FUNCTION_BLOCK FB_Logger IMPLEMENTS ZigasLibs_Core.I_LoggerEx
VAR
	_fileProperties			: ST_FileProperties;
	_logLevelHeaders		: ZigasLibs_Core.ST_LogLevelHeaders;
	_fileHandler			: FB_FileHandler;
	_logEntries				: ARRAY[0..100] OF Tc2_System.T_MaxString;
	_state					: E_LoggerState;
	_oldState				: E_LoggerState;
	_fileExists				: BOOL;
	_localSystemTime		: ZigasLibs_Core.FB_LocalSystemTimeProvider;
	_localSystemTimeString	: Tc2_System.T_MaxString;
	_stringBuilder			: ZigasLibs_Core.FB_StringBuilderBase;
	_amsAddress				: Tc2_System.ST_AmsAddr;
	_dateForLogName			: STRING;
END_VAR

_localSystemTime();
_localSystemTimeString := _localSystemTime.ConvertToString()
	.DateTime(dateSeperator := '.',
		fillWithZeros := TRUE,
		IncludeMilliseconds := FALSE,
		timeFormat := ZigasLibs_Core.E_TimeFormat.YYMMDD_HHMMSS,
		timeOfDaySeperator := ':');

IF _fileHandler.Error THEN
	_state := E_LoggerState.Error;
END_IF

CASE _state OF 
	E_LoggerState.IDLE:
		IF _logEntries[0] <> '' AND _localSystemTime.CurrentTime.IsValid THEN
			_state := E_LoggerState.WRITE_TO_FILE;
		END_IF		
		
	E_LoggerState.WRITE_TO_FILE:
		_fileHandler.FileProperties.FileLocation := _fileProperties.FileLocation;
		_fileHandler.AmsAddress.netId := AmsAddress.netId;
		_dateForLogName := _localSystemTime.ConvertToString().DateTime(
			timeFormat := ZigasLibs_Core.E_TimeFormat.YYMMDD,
			timeOfDaySeperator := '',
			dateSeperator := '',
			fillWithZeros := TRUE,
			IncludeMilliseconds := FALSE);

		_dateForLogName := _stringBuilder.Reset()
			.AddString(str := _dateForLogName)
			.AddString(str := '_')
			.AddString(str := _localSystemTime.ConvertToString().Hour(fillWithZeros := TRUE))
			.Create();
	
		_fileHandler.FileProperties.FileName := _stringBuilder.Reset()
			.AddString(str := _fileProperties.FileName)
			.AddString(str := '_')
			.AddString(str := _dateForLogName)
			.AddString(str := '.txt')
			.Create();
		
		IF NOT _fileHandler.Error AND_THEN 
			_fileHandler.WriteLine_Append(sContent := _logEntries[0]) 
		THEN
			RemoveLogEntry();
			_state := E_LoggerState.IDLE;
		END_IF
		
	E_LoggerState.ERROR:
		IF _oldState <> E_LoggerState.ERROR THEN
			_fileHandler.Reset();
		END_IF
END_CASE

_oldState := _state;

METHOD PRIVATE AddLogEntry
VAR_INPUT
	message	: Tc2_System.T_MaxString;
END_VAR

VAR
	i				: ZigasLibs_Core.T_ArrayIndexer;
	eventsMaxIndex	: ZigasLibs_Core.T_ArrayIndexer;
END_VAR
message := Tc2_Standard.CONCAT(
	STR1 := message, 
	STR2 := ZigasLibs_Core.StringConstants.NewLine);

ZigasLibs_Core.ArrayHelper.SetAtFirstEmptySlot(
	arr := _logEntries,
	item := message);
END_METHOD

{attribute 'monitoring':='variable'}
(* Gets or sets the Ams address structure*)
PROPERTY AmsAddress : REFERENCE TO ST_AmsAddr
GET
AmsAddress ref= _amsAddress;
END_GET
SET
_amsAddress := AmsAddress;
END_SET
END_PROPERTY

{attribute 'monitoring':='variable'}
PROPERTY PUBLIC BufferFull : BOOL
GET
BufferFull := _logEntries[100] <> '';
END_GET
END_PROPERTY

{attribute 'monitoring':='variable'}
(* Gets or set file properties.*)
PROPERTY FileProperties : REFERENCE TO ZigasLibs_Core.ST_FileProperties
GET
FileProperties REF= _fileProperties;
END_GET
SET
_fileProperties := FileProperties;
END_SET
END_PROPERTY

(* Logs the message without any additions.*)
METHOD LogDefault
VAR_INPUT
	message	: ZigasLibs_Core.Tc2_System.T_MaxString;
END_VAR
IF NOT Ready THEN
	RETURN;
END_IF

AddLogEntry(_stringBuilder.Reset() 
	.AddString(str := _localSystemTimeString)
	.AddString(str := ': ')
	.AddString(str := message)
	.Create());
END_METHOD

(* Logs the message by adding the error header to the start.*)
METHOD LogError
VAR_INPUT
	message	: ZigasLibs_Core.Tc2_System.T_MaxString;
END_VAR
IF NOT Ready THEN
	RETURN;
END_IF

AddLogEntry(_stringBuilder.Reset() 
	.AddString(str := _localSystemTimeString)
	.AddString(str := ': ')
	.AddString(str := _logLevelHeaders.Error)
	.AddString(str := message)
	.Create());
END_METHOD

(* Logs the message by adding the info header to the start.*)
METHOD LogInfo
VAR_INPUT
	message	: ZigasLibs_Core.Tc2_System.T_MaxString;
END_VAR
IF NOT Ready THEN
	RETURN;
END_IF

AddLogEntry(_stringBuilder.Reset() 
	.AddString(str := _localSystemTimeString)
	.AddString(str := ': ')
	.AddString(str := _logLevelHeaders.Info)
	.AddString(str := message)
	.Create());
END_METHOD

{attribute 'monitoring':='variable'}
(* Gets or sets the headers which are applied to logs for their coresponding log levels.*)
PROPERTY LogLevelHeaders : REFERENCE TO ZigasLibs_Core.ST_LogLevelHeaders
GET
LogLevelHeaders ref= _logLevelHeaders;
END_GET
SET
_logLevelHeaders := LogLevelHeaders;
END_SET
END_PROPERTY

(* Logs the message by adding the info header to the start.*)
METHOD LogWarning
VAR_INPUT
	message	: ZigasLibs_Core.Tc2_System.T_MaxString;
END_VAR
IF NOT Ready THEN
	RETURN;
END_IF

AddLogEntry(_stringBuilder.Reset() 
	.AddString(str := _localSystemTimeString)
	.AddString(str := ': ')
	.AddString(str := _logLevelHeaders.Warning)
	.AddString(str := message)
	.Create());
END_METHOD

{attribute 'monitoring':='call'}
// Returns TRUE if logger is ready to create logs. This mostly refers to system time being valid.
PROPERTY PUBLIC Ready : BOOL
GET
Ready := _localSystemTime.CurrentTime.IsValid;
END_GET
END_PROPERTY

METHOD RemoveLogEntry
ZigasLibs_Core.ArrayHelper.ShiftDown(
	arr := _logEntries, 
	dataType := _logEntries[0]);
END_METHOD

END_FUNCTION_BLOCK

(* stored: Version 1.1.0.1, ProductVersion 3.1.4024.13
   POU FB_Logger: Id {86b60fa4-cbc9-0995-00ad-63ce008210aa}, SpecialFunc None
   Method AddLogEntry: Id {6f1fe8ae-e0ba-067e-058b-4c715ea59a5c}
   Property AmsAddress: Id {2ff23ff9-8aca-06ba-18c7-b3a879ccb01f}
   Get Get: Id {87378494-b48f-041e-0273-a8548009f45b}
   Set Set: Id {03e2518e-8422-04ec-3ebc-7cb2c93733f2}
   Property BufferFull: Id {6b3f66ce-c8e6-0c2b-1325-e4b5c4b64233}
   Get Get: Id {52e4ece1-202f-0628-2423-dc2032edb2da}
   Property FileProperties: Id {673c7f63-7643-01c5-0bc9-18642143b735}
   Get Get: Id {ed145f69-492a-0c2c-1788-7460771a661c}
   Set Set: Id {80c6a351-e367-0411-01ac-b6ae657e0bcb}
   Method LogDefault: Id {03e59e35-6844-0202-3974-90f98220400a}
   Method LogError: Id {60e0135f-a63a-002e-056e-f6dc14cffeb1}
   Method LogInfo: Id {fd97ce6f-9592-08da-013c-a727bade2e2b}
   Property LogLevelHeaders: Id {4a2eeb1a-7fb2-0f80-3c56-845a85555842}
   Get Get: Id {659c25b1-4b2a-01f1-1505-fdb1e25ebd68}
   Set Set: Id {96e644fb-2cc5-081c-3f64-8981e592adf9}
   Method LogWarning: Id {76f0a31c-738d-0885-349f-e0df017a7e19}
   Property Ready: Id {c35840e3-946e-0c2d-2fef-3d51340adcda}
   Get Get: Id {19b5e194-d7eb-0906-3299-cb36db04d559}
   Method RemoveLogEntry: Id {134d7547-21a2-03bc-1ab5-77c94d18ef87} *)
